{attribute 'pack_mode' := '4'}
TYPE ST_HexMove_InitData :
STRUCT
	Header: TComInitDataHdr;
	CallByHdr: TComInitDataElmHdr;
	CallBy: TctModuleCallByType;
	ExecutionSequenceHdr: TComInitDataElmHdr;
	ExecutionSequence: TctModuleExecutionSequenceType;
	StepSizeHdr: TComInitDataElmHdr;
	StepSize: TctStepSizeType;
	ExecuteModelCodeHdr: TComInitDataElmHdr;
	ExecuteModelCode: BOOL;
	ContextInfoArr_0_TaskOidHdr: TComInitDataElmHdr;
	ContextInfoArr_0_TaskOid: OTCID;
	ContextInfoArr_0_TaskPriorityHdr: TComInitDataElmHdr;
	ContextInfoArr_0_TaskPriority: UDINT;
	ContextInfoArr_0_TaskCycleTimeNsHdr: TComInitDataElmHdr;
	ContextInfoArr_0_TaskCycleTimeNs: UDINT;
	ContextInfoArr_0_TaskPortHdr: TComInitDataElmHdr;
	ContextInfoArr_0_TaskPort: UINT;
	ContextInfoArr_0_TaskSortOrderHdr: TComInitDataElmHdr;
	ContextInfoArr_0_TaskSortOrder: UDINT;
END_STRUCT
END_TYPE

(* stored: Version 1.1.0.1, ProductVersion 3.1.4020.12
   DUT ST_HexMove_InitData: Id {9c7d0f49-5393-4f40-ab75-fdca7541fb4a} *)
